FUNCTION_BLOCK FB_HMI_STATUS
VAR_INPUT
	sText : STRING;
	stColor : T_HMI_COLORS;
END_VAR
VAR_OUTPUT
END_VAR
VAR_IN_OUT
END_VAR
VAR
END_VAR

END_FUNCTION_BLOCK

(* stored: Version 1.1.0.1, ProductVersion 3.1.4024.14
   POU FB_HMI_STATUS: Id {b6659442-3a09-4982-8e54-2e782c920cd4}, SpecialFunc None *)
